// TIA Portal V21 export
TYPE "Std_Valvola"
   STRUCT
      In : Struct
         RichiestaAutoPos : Bool;   // Richiesta di comando positivo quando in automatico
         RichiestaAutoNeg : Bool;   // Richiesta di comando negativo quando in automatico
         RichiestaAutoFolleScarico : Bool;   // Richiesta di comando scarico o folle quando in automatico
         RichiestaAutoFlipFlop : Bool;   // Richiesta di comando FLIP FLOP in automatico
         RichiestaPressionePos : Real;   // Pressione richiesta in direzione positiva (mbar)
         RichiestaPressioneNeg : Real;   // Pressione richiesta in direzione negativa (mbar)
         RichiestaPortataPos : Real;   // Portata / velocità richiesta in comando positivo (%)
         RichiestaPortataNeg : Real;   // Portata / velocità richiesta in comando negativo (%)
         ConsMovimentoPos : Bool;   // Abilitazione della valvola in direzione pos
         ConsMovimentoNeg : Bool;   // Abilitazione della valvola in direzione neg
         Feedback_SensorePos : Bool;   // Feedback di posizione digitale in positivo
         Feedback_SensoreNeg : Bool;   // Feedback di posizione digitale in negativo
         Feedback_PosizioneAttuale : Real;   // Feedback posizione attuale
         Feedback_PressionePos : Real;   // Feedback della pressione attuale mandata (mbar)
         Feedback_PressioneNeg : Real;   // Feedback della pressione attuale ritorno (mbar)
         Feedback_PortataPos : Real;   // Feedback della portata attuale mandata (mbar)
         Feedback_PortataNeg : Real;   // Feedback della portata attuale ritorno (mbar)
         Reset : Bool;
      END_STRUCT;
      Prm : Struct
         K_TipoValvola : Int;   // 0 = monostabile - 1 = bistabile
         K_VistaManuale : Int;
         TStartPos : "Std_stTimer";   // Ritardo al comando positivo
         TStopPos : "Std_stTimer";   // Ritardo alla caduta del comando positivo o al comando negativo
         TStartNeg : "Std_stTimer";   // Ritardo al comando positivo
         TStopNeg : "Std_stTimer";   // Ritardo alla caduta del comando positivo o al comando negativo
         TimeOutPos { S7_SetPoint := 'True'} : "Std_stTimer";   // Timeout posizionamento in direzione positiva
         TimeOutNeg { S7_SetPoint := 'True'} : "Std_stTimer";   // Timeout posizionamento in direzione negativa
         RitSensPos { S7_SetPoint := 'True'} : "Std_stTimer";
         RitSensNeg { S7_SetPoint := 'True'} : "Std_stTimer";
         RitFlip { S7_SetPoint := 'True'} : "Std_stTimer";
         RitFlop { S7_SetPoint := 'True'} : "Std_stTimer";
         ComportamentoTimeOut { S7_SetPoint := 'True'} : Int;   // 0 =NessunComportamento 1=TuttoPos 2=TuttoNeg 3=InvertiCmd
         MassimaPressione { S7_SetPoint := 'True'} : Int := 7000;   // mbar
         InversioneDirezione : Bool;
         TogliComandoDopoPos : Bool;   // Toglie il comando dopo aver posizionato la valvola
         SensorLess : Bool;   // DisabilitaIsensori
         UnitàMisura : "Std_UnitàDiMisura";
      END_STRUCT;
      Dati : Struct
         CondPos : Bool;   // Condizioni necessarie al comando positivo dell'uscita
         CondNeg : Bool;   // Condizioni necessarie al comando negativo dell'uscita
         RealmenteInPos : Bool;   // Fedeback valvola coerente con comando
         RealmenteInNeg : Bool;   // Fedeback valvola coerente con comando
         CmdPos : Bool;
         CmdNeg : Bool;
         BloccoRichiamato : Bool;
         InclusaInUnaSequenza : Bool;
         FlipFlop : Struct
            NumeroFlip : Struct
               Preset : Int;
               Actual : Int;
            END_STRUCT;
            MemoFlip : Bool;
            CmdFlip : Bool;
         END_STRUCT;
      END_STRUCT;
      Hmi : Struct
         StatoCmd : Struct   // Stato da popup hmi della valvola
            StatoFromHmi : Byte;   // 0=Stop 1=Auto 2=ManPos 3=ManNeg 4=Scarico
            ManPos : Bool;   // Richiesta di comando manuale positivo (Salita - Apertura - Avanti)
            ManNeg : Bool;   // Richiesta di comando manuale negativo (Discesa - Chiusura - Indietro
            ManScarico : Bool;   // Richiesta di comando manuale scarico
            Auto : Bool;   // Richiesta da HMI di rispettare le condizioni di automatico
            Stop : Bool;   // Richiesta da HMI di stop
            StatoPrecManPos : Byte;
            ManPressione : Real;   // Richiesta da HMI della pressione durante comando man
            ManPortata : Real;   // Richiesta da HMI della portata durante comando man
         END_STRUCT;
         Visibilita : Struct
            ModulantePressione : Bool;
            ModulantePortata : Bool;
            ManScarico : Bool;
            ManNegOff : Bool;
         END_STRUCT;
         RichiestaAutoPos : Bool;   // Appoggio per pulire la visualizzazione
         RichiestaAutoNeg : Bool;   // Appoggio per pulire la visualizzazione
         TipoManuale : Int;
         SiglaMeccanica : String[6];
         SiglaElettrica : String[6];
         BypassSicurezze : Bool;
      END_STRUCT;
      Allarmi : Struct
         "A" : Array[0.."K_NumAllarmiPerValvole"] of "Std_PrmAllarmeStd";
         WordHMI { S7_SetPoint := 'True'} : Word;
      END_STRUCT;
      Out : Struct
         Stato : Int;   // 0=AutoNeg / 1=Stop / 2=AutoPos / 3=ManPos / 4=ManNeg / 5=Allarme
         CmdPos : Bool;   // Uscita di comando positivo della valvola (Salita - Apertura - Avanti)
         CmdNeg : Bool;   // Uscita di comando Negativo della valvola (Discesa - Chiusura - Indietro
         CmdScarico : Bool;
         CmdPressione : Real;   // Pressione attuale (%)
         CmdPortata : Real;   // Portata / velocità attuale (%)
      END_STRUCT;
      Rif_Inc : Struct
         K_Zona : Int;
         K_Sequenza : Array[0.."K_NumRifIncrociatiSequenza"] of Int;
         K_Pid : Int;
      END_STRUCT;
   END_STRUCT;
   // // Allarmi."A"[1] : TimeOutPosiz
   // // Allarmi."A"[2] : ValvolaNonInAuto
   // // Allarmi."A"[3] : ResetRichiesto
END_TYPE
